FUNCTION ArgToIMutBinArg : Result
VAR_INPUT
	iArg		: I_Arg;
END_VAR
VAR_OUTPUT
	iVal		: I_MutBinArg;
END_VAR

IF __QUERYINTERFACE(iArg, iVal) THEN
	ArgToIMutBinArg := Ok;
END_IF

END_FUNCTION

(* stored: Version 1.1.0.1
   POU ArgToIMutBinArg: Id {9a92db2b-255b-4bd9-8710-37254a569882}, SpecialFunc None *)
